FUNCTION_BLOCK FB_2002cookie
VAR_INPUT
	execute: BOOL;
	pos2: LREAL := 2500;
END_VAR
VAR
	TIMERDONE: BOOL;
END_VAR

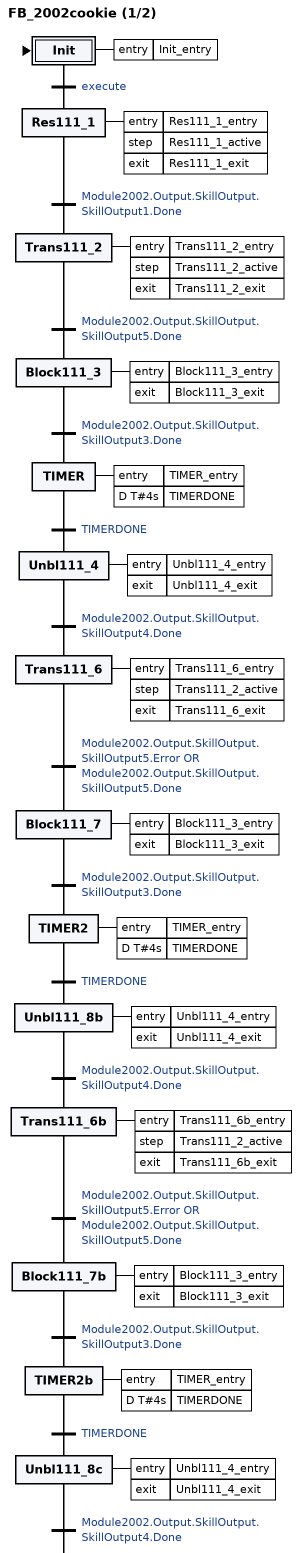
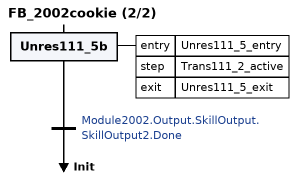
INITIAL_STEP Init:
    Init_entry(P1);  // entry action
END_STEP
TRANSITION FROM Init TO Res111_1
    := execute;
END_TRANSITION
STEP Res111_1:
    Res111_1_entry(P1);  // entry action
    Res111_1_active(N);  // step action
    Res111_1_exit(P0);  // exit action
END_STEP
TRANSITION FROM Res111_1 TO Trans111_2
    := Module2002.Output.SkillOutput.SkillOutput1.Done;
END_TRANSITION
STEP Trans111_2:
    Trans111_2_entry(P1);  // entry action
    Trans111_2_active(N);  // step action
    Trans111_2_exit(P0);  // exit action
END_STEP
TRANSITION FROM Trans111_2 TO Block111_3
    := Module2002.Output.SkillOutput.SkillOutput5.Done;
END_TRANSITION
STEP Block111_3:
    Block111_3_entry(P1);  // entry action
    Block111_3_exit(P0);  // exit action
END_STEP
TRANSITION FROM Block111_3 TO TIMER
    := Module2002.Output.SkillOutput.SkillOutput3.Done;
END_TRANSITION
STEP TIMER:
    TIMER_entry(P1);  // entry action
    TIMERDONE(D, T#4s);
END_STEP
TRANSITION FROM TIMER TO Unbl111_4
    := TIMERDONE;
END_TRANSITION
STEP Unbl111_4:
    Unbl111_4_entry(P1);  // entry action
    Unbl111_4_exit(P0);  // exit action
END_STEP
TRANSITION FROM Unbl111_4 TO Trans111_6
    := Module2002.Output.SkillOutput.SkillOutput4.Done;
END_TRANSITION
STEP Trans111_6:
    Trans111_6_entry(P1);  // entry action
    Trans111_2_active(N);  // step action
    Trans111_6_exit(P0);  // exit action
END_STEP
TRANSITION FROM Trans111_6 TO Block111_7
    := Module2002.Output.SkillOutput.SkillOutput5.Error OR Module2002.Output.SkillOutput.SkillOutput5.Done;
END_TRANSITION
STEP Block111_7:
    Block111_3_entry(P1);  // entry action
    Block111_3_exit(P0);  // exit action
END_STEP
TRANSITION FROM Block111_7 TO TIMER2
    := Module2002.Output.SkillOutput.SkillOutput3.Done;
END_TRANSITION
STEP TIMER2:
    TIMER_entry(P1);  // entry action
    TIMERDONE(D, T#4s);
END_STEP
TRANSITION FROM TIMER2 TO Unbl111_8b
    := TIMERDONE;
END_TRANSITION
STEP Unbl111_8b:
    Unbl111_4_entry(P1);  // entry action
    Unbl111_4_exit(P0);  // exit action
END_STEP
TRANSITION FROM Unbl111_8b TO Trans111_6b
    := Module2002.Output.SkillOutput.SkillOutput4.Done;
END_TRANSITION
STEP Trans111_6b:
    Trans111_6b_entry(P1);  // entry action
    Trans111_2_active(N);  // step action
    Trans111_6b_exit(P0);  // exit action
END_STEP
TRANSITION FROM Trans111_6b TO Block111_7b
    := Module2002.Output.SkillOutput.SkillOutput5.Error OR Module2002.Output.SkillOutput.SkillOutput5.Done;
END_TRANSITION
STEP Block111_7b:
    Block111_3_entry(P1);  // entry action
    Block111_3_exit(P0);  // exit action
END_STEP
TRANSITION FROM Block111_7b TO TIMER2b
    := Module2002.Output.SkillOutput.SkillOutput3.Done;
END_TRANSITION
STEP TIMER2b:
    TIMER_entry(P1);  // entry action
    TIMERDONE(D, T#4s);
END_STEP
TRANSITION FROM TIMER2b TO Unbl111_8c
    := TIMERDONE;
END_TRANSITION
STEP Unbl111_8c:
    Unbl111_4_entry(P1);  // entry action
    Unbl111_4_exit(P0);  // exit action
END_STEP
TRANSITION FROM Unbl111_8c TO Unres111_5b
    := Module2002.Output.SkillOutput.SkillOutput4.Done;
END_TRANSITION
STEP Unres111_5b:
    Unres111_5_entry(P1);  // entry action
    Trans111_2_active(N);  // step action
    Unres111_5_exit(P0);  // exit action
END_STEP
TRANSITION FROM Unres111_5b TO Init
    := Module2002.Output.SkillOutput.SkillOutput2.Done;
END_TRANSITION

ACTION Res111_1_entry:
// Reservieren entry
Module2002.Input.SkillInput.SkillInput1.Execute := TRUE;
Module2002.Input.SkillInput.SkillInput1.ParameterInput.Parameterinput1.Value := 112; //TASKID
END_ACTION

ACTION Unbl111_4_exit:
//unBLOCKIEREN

Module2002.Input.SkillInput.SkillInput4.Execute := FALSE; 
Module2002.Input.SkillInput.SkillInput4.ParameterInput.Parameterinput1.Value := 000; //TaskID
END_ACTION

ACTION Trans111_6b_exit:
//TRANSPORTIEREN

Module2002.Input.SkillInput.SkillInput5.Execute := FALSE;
Module2002.Input.SkillInput.SkillInput5.ParameterInput.Parameterinput1.Value := 0; //X-Position
Module2002.Input.SkillInput.SkillInput5.ParameterInput.Parameterinput2.Value := 0; //Z-Position
Module2002.Input.SkillInput.SkillInput5.ParameterInput.Parameterinput3.Value := 0; //Velocity
Module2002.Input.SkillInput.SkillInput5.ParameterInput.Parameterinput4.Value := 0; //Acceleration
END_ACTION

ACTION Res111_1_active:

END_ACTION

ACTION Trans111_2_entry_1:
//TRANSPORTIEREN

Module2002.Input.SkillInput.SkillInput5.Execute := TRUE;
Module2002.Input.SkillInput.SkillInput5.ParameterInput.Parameterinput1.Value := 3000; //X-Position
Module2002.Input.SkillInput.SkillInput5.ParameterInput.Parameterinput2.Value := 0; //Z-Position
Module2002.Input.SkillInput.SkillInput5.ParameterInput.Parameterinput3.Value := 0; //Velocity
Module2002.Input.SkillInput.SkillInput5.ParameterInput.Parameterinput4.Value := 0; //Acceleration
END_ACTION

ACTION Unres111_5_entry:
//unreserve
Module2002.Input.SkillInput.SkillInput2.Execute := TRUE;
Module2002.Input.SkillInput.SkillInput2.ParameterInput.Parameterinput1.Value := 112; //TaskID
END_ACTION

ACTION Block111_3_exit:
//BLOCKIEREN

Module2002.Input.SkillInput.SkillInput3.Execute := FALSE;
Module2002.Input.SkillInput.SkillInput3.ParameterInput.Parameterinput1.Value := 0; //TaskID
END_ACTION

ACTION Trans111_6_exit:
//TRANSPORTIEREN

Module2002.Input.SkillInput.SkillInput5.Execute := FALSE;
Module2002.Input.SkillInput.SkillInput5.ParameterInput.Parameterinput1.Value := 0; //X-Position
Module2002.Input.SkillInput.SkillInput5.ParameterInput.Parameterinput2.Value := 0; //Z-Position
Module2002.Input.SkillInput.SkillInput5.ParameterInput.Parameterinput3.Value := 0; //Velocity
Module2002.Input.SkillInput.SkillInput5.ParameterInput.Parameterinput4.Value := 0; //Acceleration
END_ACTION

ACTION Unbl111_4_entry:
//unBLOCKIEREN

Module2002.Input.SkillInput.SkillInput4.Execute := TRUE; //FALSE weil timer
Module2002.Input.SkillInput.SkillInput4.ParameterInput.Parameterinput1.Value := 112; //TaskID
END_ACTION

ACTION TIMER_entry:
TIMERDONE := FALSE;
END_ACTION

ACTION Trans111_2_entry:
//TRANSPORTIEREN

Module2002.Input.SkillInput.SkillInput5.Execute := TRUE;
Module2002.Input.SkillInput.SkillInput5.ParameterInput.Parameterinput1.Value := 3000; //X-Position
Module2002.Input.SkillInput.SkillInput5.ParameterInput.Parameterinput2.Value := 0; //Z-Position
Module2002.Input.SkillInput.SkillInput5.ParameterInput.Parameterinput3.Value := 0; //Velocity
Module2002.Input.SkillInput.SkillInput5.ParameterInput.Parameterinput4.Value := 0; //Acceleration
END_ACTION

ACTION Trans111_6_entry:
//TRANSPORTIEREN

Module2002.Input.SkillInput.SkillInput5.Execute := TRUE;
Module2002.Input.SkillInput.SkillInput5.ParameterInput.Parameterinput1.Value := 3400; //X-Position
Module2002.Input.SkillInput.SkillInput5.ParameterInput.Parameterinput2.Value := 80; //Z-Position
Module2002.Input.SkillInput.SkillInput5.ParameterInput.Parameterinput3.Value := 0; //Velocity
Module2002.Input.SkillInput.SkillInput5.ParameterInput.Parameterinput4.Value := 0; //Acceleration
END_ACTION

ACTION Res111_1_exit:
// Reservieren entry
Module2002.Input.SkillInput.SkillInput1.Execute := FALSE;
Module2002.Input.SkillInput.SkillInput1.ParameterInput.Parameterinput1.Value := 0; //TASKID
END_ACTION

ACTION Trans111_2_exit:
//TRANSPORTIEREN

Module2002.Input.SkillInput.SkillInput5.Execute := FALSE;
Module2002.Input.SkillInput.SkillInput5.ParameterInput.Parameterinput1.Value := 0; //X-Position
Module2002.Input.SkillInput.SkillInput5.ParameterInput.Parameterinput2.Value := 0; //Z-Position
Module2002.Input.SkillInput.SkillInput5.ParameterInput.Parameterinput3.Value := 0; //Velocity
Module2002.Input.SkillInput.SkillInput5.ParameterInput.Parameterinput4.Value := 0; //Acceleration
END_ACTION

ACTION Init_entry:
execute := FALSE;
END_ACTION

ACTION Trans111_2_active:

END_ACTION

ACTION Trans111_6b_entry:
Module2002.Input.SkillInput.SkillInput5.Execute := TRUE;
Module2002.Input.SkillInput.SkillInput5.ParameterInput.Parameterinput1.Value := 3000; //X-Position
Module2002.Input.SkillInput.SkillInput5.ParameterInput.Parameterinput2.Value := 80; //Z-Position
Module2002.Input.SkillInput.SkillInput5.ParameterInput.Parameterinput3.Value := 0; //Velocity
Module2002.Input.SkillInput.SkillInput5.ParameterInput.Parameterinput4.Value := 0; //Acceleration
END_ACTION

ACTION Block111_3_entry:
//BLOCKIEREN

Module2002.Input.SkillInput.SkillInput3.Execute := TRUE;
Module2002.Input.SkillInput.SkillInput3.ParameterInput.Parameterinput1.Value := 112; //TaskID
END_ACTION

ACTION Unres111_5_exit:
//unreserve
Module2002.Input.SkillInput.SkillInput2.Execute := FALSE;
Module2002.Input.SkillInput.SkillInput2.ParameterInput.Parameterinput1.Value := 0; //TaskID
END_ACTION

END_FUNCTION_BLOCK

(* stored: Version 1.1.0.1, ProductVersion 3.1.0.25
   POU FB_2002cookie: Id {520c64b7-644c-4f65-9e42-59bcd0a24c81}
   Action Res111_1_entry: Id {01c98250-ee6c-41cd-b651-c651d0d4965e}
   Action Unbl111_4_exit: Id {04a979b0-0ff6-4287-977b-2569506a5f1d}
   Action Trans111_6b_exit: Id {0d24c0c9-2ec8-4e4e-b3af-3d7e7c070a6f}
   Action Res111_1_active: Id {1768219b-0478-4836-bd5a-4d3b76ee47de}
   Action Trans111_2_entry_1: Id {1a0fcbbe-9a0f-4713-83c6-e723e13cba07}
   Action Unres111_5_entry: Id {276624e7-d7de-453d-aff2-c2fcd711cfb0}
   Action Block111_3_exit: Id {2e7f8998-ae1b-4bfe-bbb6-6683b856c764}
   Action Trans111_6_exit: Id {34eb1791-0a4f-4984-8210-0fe25984836e}
   Action Unbl111_4_entry: Id {38f982ae-5bbc-4fee-a7ad-81f6235bb476}
   Action TIMER_entry: Id {3aaf2434-1ed1-4d78-be9a-7ff61c89f6de}
   Action Trans111_2_entry: Id {49551371-78f5-4b20-8649-cf4dd0f94f30}
   Action Trans111_6_entry: Id {887eb957-ee77-410e-968c-0ea634f330ed}
   Action Res111_1_exit: Id {90117419-94ec-4be7-b436-646c00ca51f9}
   Action Trans111_2_exit: Id {9b878f25-dec0-46b4-a35f-c17a1b8e7516}
   Action Init_entry: Id {a1696bf4-a8d9-4ba4-b88e-de8e606b73eb}
   Action Trans111_2_active: Id {b0464620-bda5-4c95-b912-08b2939b7c34}
   Action Trans111_6b_entry: Id {d92cd585-a354-4a3b-92f6-10b085e0b2b1}
   Action Block111_3_entry: Id {f798a510-e41b-4878-aedc-390766f99f25}
   Action Unres111_5_exit: Id {fef7f832-5de3-488c-aa3a-eac70c3cdea4} *)
